(* CODESYS project IceMaker.xml

Project tree, tasks and I/O mapping:
  function block IceMaker [CFC]
*)

// IceMaker
FUNCTION_BLOCK IceMaker
//  .					.					.
VAR_INPUT
	Enable: 			BOOL;
	NeedIce: 			BOOL;
	StirComplete: 		BOOL;
	MakeIceTimeout: 	TIME;
	FaultReset: 		BOOL;
	MakeIceOverride:	BOOL;
END_VAR
VAR_OUTPUT
	StirIce: 			BOOL;
	MakeIce: 			BOOL;
	Fault: 				BOOL;
END_VAR
VAR
	_Sequence: IceMakerSequence;
	_ManualFaultReset: BOOL;
	_MakeIceFault: BOOL;
END_VAR
//  .					.					.
//  Ice Maker Maintenance Page HMI Elements
//  Element				Type				Tag
//  ------------------------------------------------------------------
//  Enable				Toggle				Settings.IceMaker.Enable
//  Timeout				Numeric				Settings.IceMaker.MakeIceTimeout
//  Need Ice			Bit Lamp			Components.IceMaker.NeedIce
//  Make Ice			Bit Lamp			Components.IceMaker.MakeIce
//  Make Ice Override	Toggle				Settings.IceMaker.MakeIceOverride
//  Stir Ice			Bit Lamp			Components.IceMaker.StirIce
//  Make Ice Fault		Bit Lamp			Components.IceMaker.MakeIceFault
//  Fault Reset			Button				Components.IceMaker._ManualFaultReset
// 
//  Outside Component Maintenance Page HMI Elements
//  Ice Level Okay		Bit Lamp			Components.Hopper.IceLevelOkay
//  Agitating			Bit Lamp			Components.Agitator.Agitating
VAR // added by the converter: edge detectors and wires of the graphical bodies
    _w1 : BOOL;
END_VAR

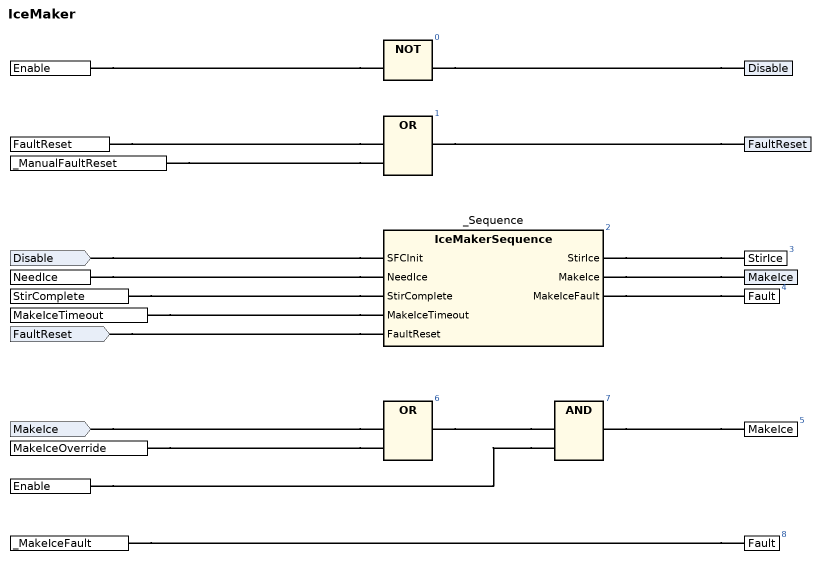
_Sequence(
    SFCInit := NOT Enable,
    NeedIce := NeedIce,
    StirComplete := StirComplete,
    MakeIceTimeout := MakeIceTimeout,
    FaultReset := FaultReset OR _ManualFaultReset); // IceMakerSequence
StirIce := _Sequence.StirIce;
Fault := _Sequence.MakeIceFault;
MakeIce := _w1;
_w1 := (_Sequence.MakeIce OR MakeIceOverride) AND Enable;
Fault := _MakeIceFault;

END_FUNCTION_BLOCK
